{attribute 'qualified_only'}
VAR_GLOBAL
	//Controls I/O
	bHomeLampBlueState 	: BOOL;
	
	//Indicators
	
	//Cycle Control
	bBtStartCycle		: BOOL := FALSE; //Button Start Cycle from HMI
	bBtStopCycle		: BOOL := FALSE; //Button Start Cycle from HMI
	
END_VAR

(* stored: Version 1.1.0.1, ProductVersion 3.1.4024.12
   GVL GVL_HMIVariables: Id {0409f918-eea3-4325-9608-40b83ff788af} *)
